FUNCTION_BLOCK ControlFunc
VAR_OUTPUT
	Active : BOOL;
END_VAR
VAR CONSTANT
	AXIS_MIN_IDX : USINT := 1;
	AXIS_MAX_IDX : USINT := 6;
END_VAR
VAR
	idx : USINT(AXIS_MIN_IDX..AXIS_MAX_IDX);
	
	state : ST_6Axis_State;
	command : E_6Axis_Command;
	
	Axis : ARRAY[AXIS_MIN_IDX..AXIS_MAX_IDX] OF AXIS_REF;
	Power : ARRAY[AXIS_MIN_IDX..AXIS_MAX_IDX] OF MC_Power;
	Stop : ARRAY[AXIS_MIN_IDX..AXIS_MAX_IDX] OF MC_Stop;
	Halt : ARRAY[AXIS_MIN_IDX..AXIS_MAX_IDX] OF MC_Halt; //delete
	AbsPos : ARRAY[AXIS_MIN_IDX..AXIS_MAX_IDX] OF MC_MoveAbsolute;
	ExtSwitchEn : ARRAY[AXIS_MIN_IDX..AXIS_MAX_IDX] OF MC_ExtSetPointGenEnable;
	ExtSwitchDis : ARRAY[AXIS_MIN_IDX..AXIS_MAX_IDX] OF MC_ExtSetPointGenDisable;
	KM : Kinematics;
	//fb_line : ExtLine;
	
	HomeAngles : ARRAY[AXIS_MIN_IDX..AXIS_MAX_IDX] OF DINT := [0, 0, 0, 0, 0, 0];
	JointDegNow : ARRAY[AXIS_MIN_IDX..AXIS_MAX_IDX] OF LREAL;
	xyzNow : ARRAY[1..3] OF LREAL;
	rpyNow : ARRAY[1..3] OF LREAL;
	
	
	

	TestPos : ARRAY[AXIS_MIN_IDX..AXIS_MAX_IDX] OF LREAL := [450, -15, 290, 137, 0, 0];
	angles : ARRAY[1..6] OF LREAL; 
	
	
	
END_VAR

readAxis();

CASE command OF
	E_6Axis_Command.NO_COMMAND:
		FOR idx := AXIS_MIN_IDX TO AXIS_MAX_IDX DO
			AbsPos[idx].Execute := FALSE;
			
		END_FOR
		
	E_6Axis_Command.POWER_ON:
		FOR idx := AXIS_MIN_IDX TO AXIS_MAX_IDX DO
			Power[idx].Enable := TRUE;
		END_FOR
		IF state.powerOn THEN
			command := E_6Axis_Command.HOMING;
		END_IF
	
	E_6Axis_Command.HOMING:
		FOR idx := AXIS_MIN_IDX TO AXIS_MAX_IDX DO	
			AbsPos[idx].Execute := TRUE;
			AbsPos[idx].Position := HomeAngles[idx];
			AbsPos[idx].Velocity := 5;
		END_FOR
		IF NOT state.moving AND AbsPos[1].Done AND AbsPos[2].Done AND AbsPos[3].Done AND AbsPos[4].Done  AND AbsPos[5].Done AND AbsPos[6].Done THEN
			command := E_6axis_Command.NO_COMMAND;	
		END_IF
		
		
	E_6Axis_Command.PTP:
		KM.Inverse(position := TestPos, angles => angles);
		FOR idx := AXIS_MIN_IDX TO AXIS_MAX_IDX DO	
			AbsPos[idx].Execute := TRUE;
			AbsPos[idx].Position := angles[idx];
			AbsPos[idx].Velocity := 5;
		END_FOR
		
		IF NOT state.moving AND AbsPos[1].Done AND AbsPos[2].Done AND AbsPos[3].Done AND AbsPos[4].Done  AND AbsPos[5].Done AND AbsPos[6].Done THEN
			command := E_6axis_Command.NO_COMMAND;	
		END_IF
		
		
		

END_CASE

ActMove();
ActPower();
ActStop();

ACTION ActExternalMove:
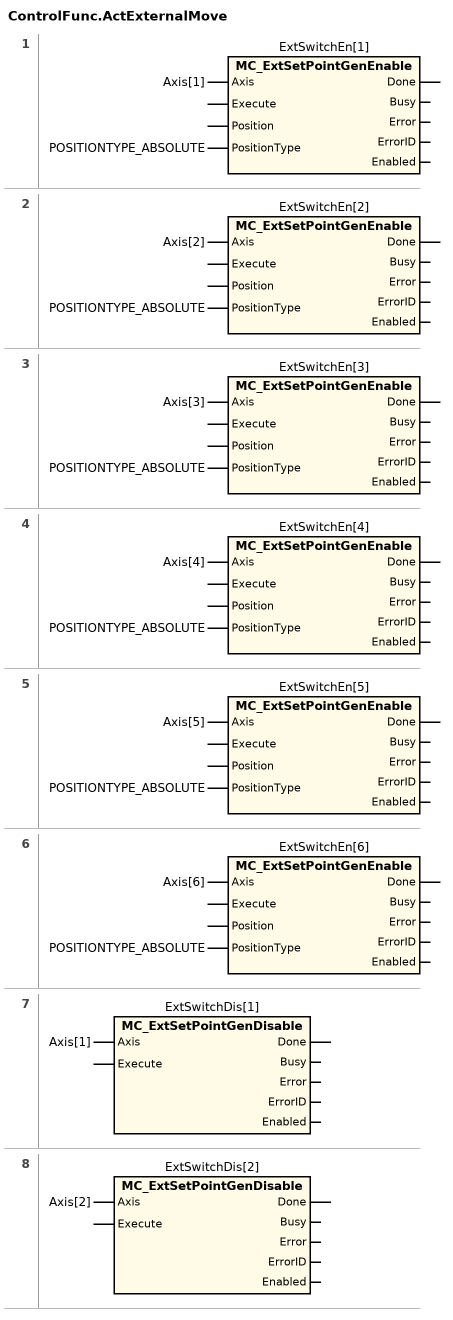
// NETWORK 1
ExtSwitchEn[1](Axis := Axis[1], PositionType := POSITIONTYPE_ABSOLUTE); // MC_ExtSetPointGenEnable

// NETWORK 2
ExtSwitchEn[2](Axis := Axis[2], PositionType := POSITIONTYPE_ABSOLUTE); // MC_ExtSetPointGenEnable

// NETWORK 3
ExtSwitchEn[3](Axis := Axis[3], PositionType := POSITIONTYPE_ABSOLUTE); // MC_ExtSetPointGenEnable

// NETWORK 4
ExtSwitchEn[4](Axis := Axis[4], PositionType := POSITIONTYPE_ABSOLUTE); // MC_ExtSetPointGenEnable

// NETWORK 5
ExtSwitchEn[5](Axis := Axis[5], PositionType := POSITIONTYPE_ABSOLUTE); // MC_ExtSetPointGenEnable

// NETWORK 6
ExtSwitchEn[6](Axis := Axis[6], PositionType := POSITIONTYPE_ABSOLUTE); // MC_ExtSetPointGenEnable

// NETWORK 7
ExtSwitchDis[1](Axis := Axis[1]); // MC_ExtSetPointGenDisable

// NETWORK 8
ExtSwitchDis[2](Axis := Axis[2]); // MC_ExtSetPointGenDisable

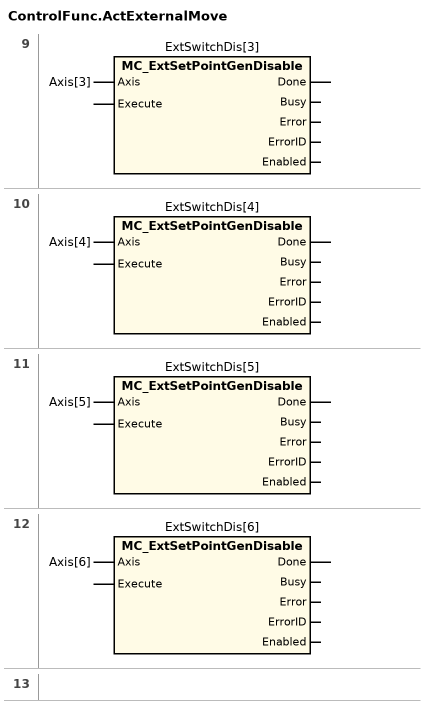
// NETWORK 9
ExtSwitchDis[3](Axis := Axis[3]); // MC_ExtSetPointGenDisable

// NETWORK 10
ExtSwitchDis[4](Axis := Axis[4]); // MC_ExtSetPointGenDisable

// NETWORK 11
ExtSwitchDis[5](Axis := Axis[5]); // MC_ExtSetPointGenDisable

// NETWORK 12
ExtSwitchDis[6](Axis := Axis[6]); // MC_ExtSetPointGenDisable

// NETWORK 13
END_ACTION

ACTION ActMove:
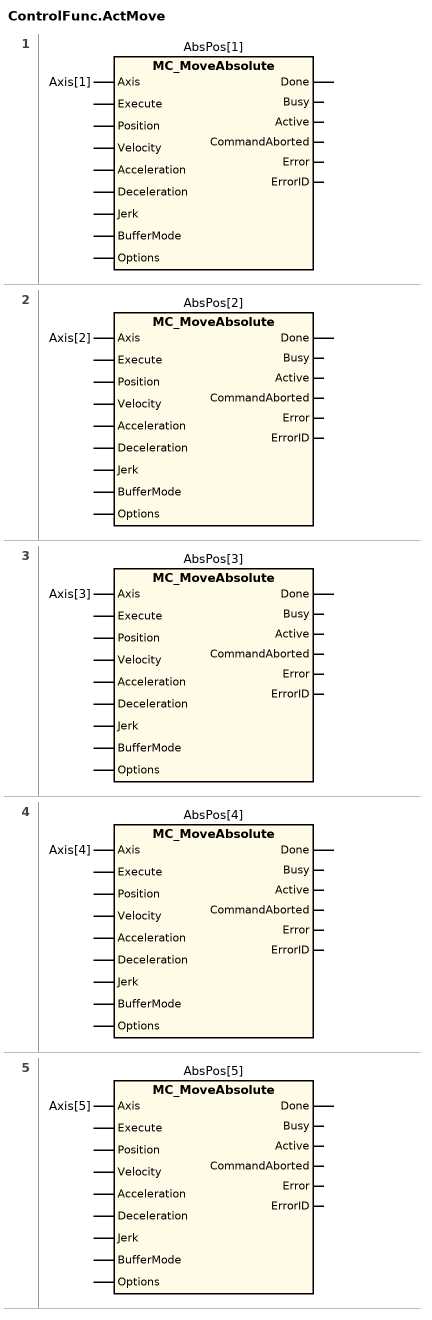
// NETWORK 1
AbsPos[1](Axis := Axis[1]); // MC_MoveAbsolute

// NETWORK 2
AbsPos[2](Axis := Axis[2]); // MC_MoveAbsolute

// NETWORK 3
AbsPos[3](Axis := Axis[3]); // MC_MoveAbsolute

// NETWORK 4
AbsPos[4](Axis := Axis[4]); // MC_MoveAbsolute

// NETWORK 5
AbsPos[5](Axis := Axis[5]); // MC_MoveAbsolute

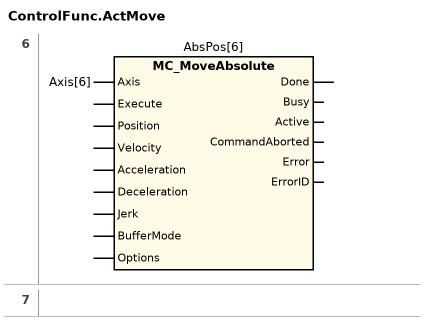
// NETWORK 6
AbsPos[6](Axis := Axis[6]); // MC_MoveAbsolute

// NETWORK 7
END_ACTION

ACTION ActPower:
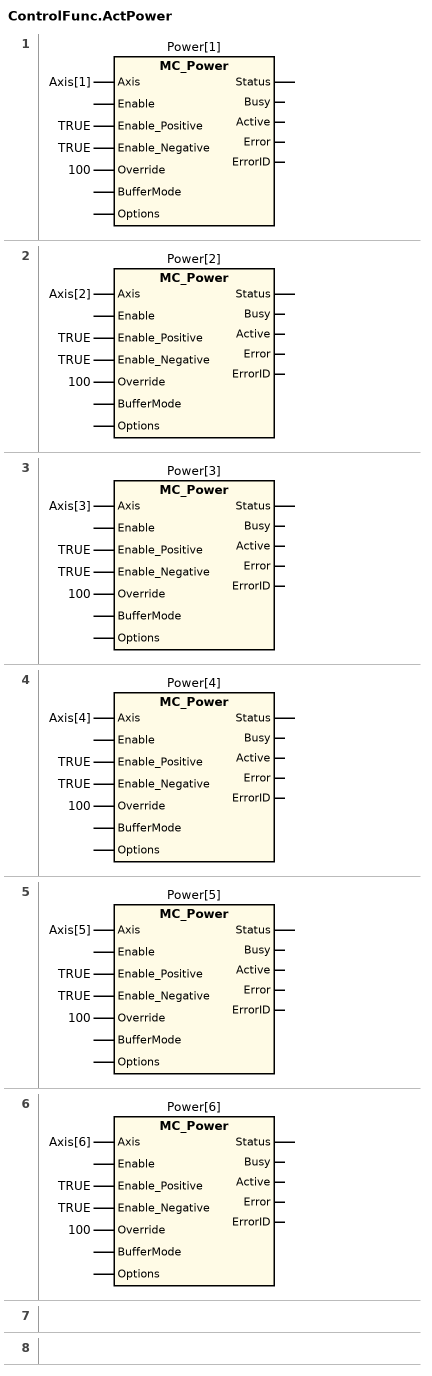
// NETWORK 1
Power[1](Axis := Axis[1], Enable_Positive := TRUE, Enable_Negative := TRUE, Override := 100); // MC_Power

// NETWORK 2
Power[2](Axis := Axis[2], Enable_Positive := TRUE, Enable_Negative := TRUE, Override := 100); // MC_Power

// NETWORK 3
Power[3](Axis := Axis[3], Enable_Positive := TRUE, Enable_Negative := TRUE, Override := 100); // MC_Power

// NETWORK 4
Power[4](Axis := Axis[4], Enable_Positive := TRUE, Enable_Negative := TRUE, Override := 100); // MC_Power

// NETWORK 5
Power[5](Axis := Axis[5], Enable_Positive := TRUE, Enable_Negative := TRUE, Override := 100); // MC_Power

// NETWORK 6
Power[6](Axis := Axis[6], Enable_Positive := TRUE, Enable_Negative := TRUE, Override := 100); // MC_Power

// NETWORK 7

// NETWORK 8
END_ACTION

ACTION ActStop:
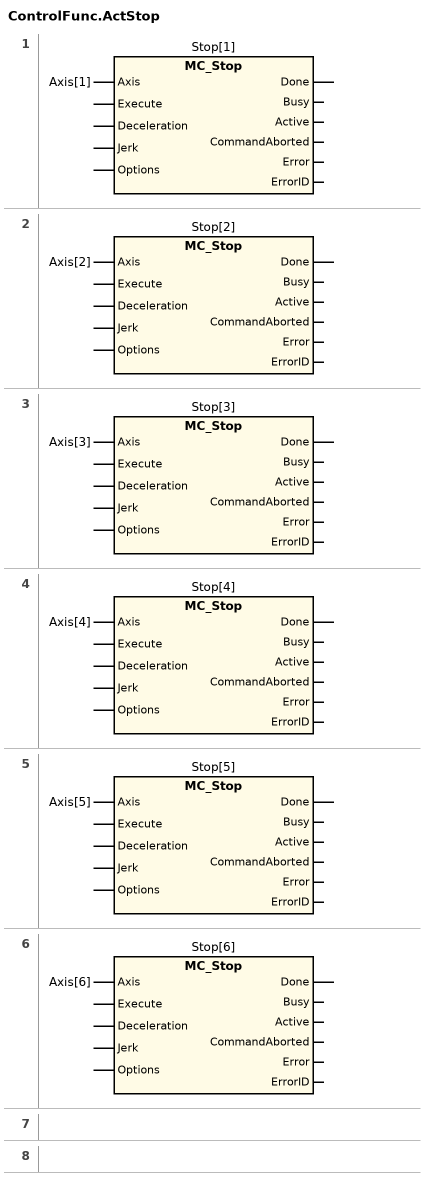
// NETWORK 1
Stop[1](Axis := Axis[1]); // MC_Stop

// NETWORK 2
Stop[2](Axis := Axis[2]); // MC_Stop

// NETWORK 3
Stop[3](Axis := Axis[3]); // MC_Stop

// NETWORK 4
Stop[4](Axis := Axis[4]); // MC_Stop

// NETWORK 5
Stop[5](Axis := Axis[5]); // MC_Stop

// NETWORK 6
Stop[6](Axis := Axis[6]); // MC_Stop

// NETWORK 7

// NETWORK 8
END_ACTION

METHOD CalculatePath : BOOL

VAR_INPUT
	final_pos : ARRAY [1..6] OF LREAL;
END_VAR

VAR 
	xyz : ARRAY [1..3] OF LREAL;
	rpy : ARRAY [1..3] OF LREAL;

END_VAR
END_METHOD

METHOD move_PTP : BOOL

VAR_INPUT
	// position : [x, y, z, r, p, y]
	position : ARRAY[1..6] OF LREAL; 
	executeTime : LREAL;
END_VAR

VAR
	idx : USINT;
	msg : ST_Msg_PTP;
END_VAR
END_METHOD

METHOD readAxis : BOOL

VAR
	PositionNow : ARRAY[1..6] OF LREAL;
	
END_VAR
FOR idx := AXIS_MIN_IDX TO AXIS_MAX_IDX DO
	Axis[idx]();
	JointDegNow[idx] := Axis[idx].NcToPlc.ActPos;
END_FOR
KM.Forward(angles := JointDegNow, position => PositionNow);
FOR idx := 1 TO 3 DO
	xyzNow[idx] := PositionNow[idx];
	rpyNow[idx] := PositionNow[idx+3];
END_FOR

state.powerOn := Power[1].Status AND Power[2].Status AND Power[3].Status AND Power[4].Status AND Power[5].Status AND Power[6].Status;
state.stop := Stop[1].Done AND Stop[2].Done AND Stop[3].Done AND Stop[4].Done AND Stop[5].Done AND Stop[6].Done;
state.moving := Axis[1].Status.Moving OR Axis[2].Status.Moving OR Axis[3].Status.Moving OR  Axis[4].Status.Moving OR Axis[5].Status.Moving OR Axis[6].Status.Moving;
//state.pause := NOT (state.moving OR state.stop);
state.error := Axis[1].Status.Error OR Axis[2].Status.Error OR Axis[3].Status.Error OR Axis[4].Status.Error OR Axis[5].Status.Error OR Axis[6].Status.Error;
//state.ready := Axis[1].Status.Operational AND Axis[2].Status.Operational AND Axis[3].Status.Operational AND Axis[4].Status.Operational AND Axis[5].Status.Operational AND Axis[6].Status.Operational;
END_METHOD

END_FUNCTION_BLOCK

(* stored: Version 1.1.0.1, ProductVersion 3.1.4024.12
   POU ControlFunc: Id {d85eeb7a-7828-4eea-9de8-5b49fe19e8b9}, SpecialFunc None
   Action ActExternalMove: Id {3582fa84-2718-4e34-b3be-b419c476ca0a}
   Action ActMove: Id {0fa0cb91-03cb-4036-87db-d890a57ebb64}
   Action ActPower: Id {c3eeae36-d769-4e1a-aa08-55704f8ad648}
   Action ActStop: Id {64d4d7a6-ae28-4a6a-8a4f-bf6b60852155}
   Method CalculatePath: Id {8afb4caa-dc5e-4451-b03d-00b3003892e3}
   Method move_PTP: Id {d91d5db4-9583-48ea-8990-a124e50c5070}
   Method readAxis: Id {ba379574-a876-4daa-b1b9-555b1a112c69} *)
